// TwinCAT 3 PLC project Valve_AutoCalibration
// ProgramVersion: 3.1.4023.0
// libraries:
//   Tc2_Standard, * (Beckhoff Automation GmbH)
//   Tc2_System, * (Beckhoff Automation GmbH)
//   Tc3_Module, * (Beckhoff Automation GmbH)
// project tree:
//   / PlcTask.TcTTO
//   POUs/AutoCalibrate/ FB_AutoCalibration.TcPOU, FB_OnSetpointCheck.TcPOU, FB_PulseGen.TcPOU
//   POUs/ MAIN.TcPOU
// real-time tasks:
//   TASK PlcTask: cycle T#10ms, priority 20, ADS port 350

CONFIGURATION Valve_AutoCalibration
    RESOURCE PLC ON TwinCAT3
        TASK PlcTask(INTERVAL := T#10ms, PRIORITY := 20);
        PROGRAM MAIN WITH PlcTask : MAIN;
    END_RESOURCE
END_CONFIGURATION

// ---- POUs/MAIN.TcPOU
PROGRAM MAIN
VAR
bCalibrate:	BOOL;
fFB: REAL;
fStepValue: REAL :=0.5;
fDev: REAL := 0.1;	
fCmd: REAL;
fCommandZeroError:	REAL;
fCommandSpanError:	REAL;
fFeedbackZeroError:	REAL;
fFeedbackSpanError: REAL;  
bCalibrationFinished: BOOL;
bError : BOOL;
bBusy : BOOL;
bDoubleCheck : BOOL;
fbAutoCalibration : FB_AutoCalibration;
END_VAR

fbAutoCalibration(bCalibrate:=bCalibrate,
				fFB := fFB,
				fStepValue:=fStepValue,
				fDev:=fDev,
				fBand:=0.2);

fCmd:= fbAutoCalibration.fCmd;
				
fCommandZeroError:= fbAutoCalibration.fCmdZeroErr;

fCommandSpanError:= fbAutoCalibration.fCmdSpanErr;

fFeedbackZeroError:= fbAutoCalibration.fFBZeroErr;

fFeedbackSpanError:= fbAutoCalibration.fFBSpanErr;

bCalibrationFinished:=fbAutoCalibration.bCalibrationFinished;

bError := fbAutoCalibration.bError;

bBusy := fbAutoCalibration.bBusy;

bDoubleCheck := fbAutoCalibration.bDoubleCheck;

END_PROGRAM

// ---- POUs/AutoCalibrate/FB_AutoCalibration.TcPOU
FUNCTION_BLOCK FB_AutoCalibration
VAR_INPUT	
	bCalibrate:	BOOL; 	 //Calibration is ON
	fFB: REAL;			 //Valve feedback
	fStepValue: REAL;	 //Step value for the control valve
	fDev: REAL;			 //Deviation value to be catched in the feedback signal after the control valve stepped up
	fBand: REAL;		 //Acceptable deviation in the feedback for the double check
END_VAR
VAR_OUTPUT
	fCmd: REAL;					//Valve control signal
	fCmdZeroErr: REAL;			//Control singal zero error
	fCmdSpanErr: REAL;			//Control singal span error
	fFBZeroErr:	REAL;			//Feedback signal zero error
	fFBSpanErr: REAL;  			//Feedback span error	
	bCalibrationFinished: BOOL;	//Calibration completed
	bDoubleCheck: BOOL;			//True: Double check succesfful, FALSE: Double check failed 
	bBusy: BOOL;				//Calibration is working
	bError: BOOL;				//Error, if the valve does not open, close or exceeds the min/max values
END_VAR
VAR	
	bZeroErrCalibComplet: BOOL;
	bSpanErrCalibComplet: BOOL;
	fbPulseGenZeroErr : FB_PulseGen;
	fbPulseGenSpanErr : FB_PulseGen;
	fCmdPrevState : REAL;
	fFBPrevState : REAL;	
	RTrigCalibON : R_TRIG;	
	RTrigZero : R_TRIG;
	RTrigSpan : R_TRIG;
	bValveClosed : BOOL;
	bValveOpened : BOOL;
	bDoubleCheckFail  : BOOL;
	_fbTimerValveClosing: TON;
	_fbTimerValveOpening : TON;
	_bClosingTimer : BOOL;	
	_bOpeningTimer : BOOL;	
	_fbTimerDoubleCheck : TON;
	_bTimerDoubleCheck : BOOL;	
	_fbTimerOnMinFB	: TON;
	_fbTimerOnMaxFB	: TON;
	_bMinFBChecked : BOOL;
	_bMaxFBChecked : BOOL;
END_VAR
VAR CONSTANT
	fMinPos: REAL := 0.0;
	fMaxPos: REAL := 100.0;
	tPtON: TIME := T#0.01S;
	tPtOFF: TIME := T#5S;
	_tCloseValve: TIME := T#20S;		//20 seconds for closing the valve
	_tOpenValve: TIME := T#120S;		//120 seconds for opening the valve
	_fMinFB: REAL := 3.0;				//Min Input signal 4mA +- %2
	_fMaxFB: REAL := 96.04;				//Max Input signal 19.6mA +- %2
	_tDoubleCheck : TIME := T#150S;		//Max time for completing the double check (120s opening + 20s closing + 10s on FB check)	
	_tDelay : TIME := T#5S;				//Time for on setpoint check
END_VAR

//Initialization for the next calibration cycle
RTrigCalibON(CLK:= bCalibrate);
IF RTrigCalibON.Q AND NOT bBusy THEN		
	fFBPrevState := fFB;	
	fCmdZeroErr:= 0.0;
	fCmdSpanErr:= 0.0;
	fFBZeroErr:= 0.0;
	fFBSpanErr:= 0.0;
	bDoubleCheck:= FALSE;
	bDoubleCheckFail:= FALSE;
	bError := FALSE;	
	bBusy := TRUE;		
	bZeroErrCalibComplet := FALSE;
	bSpanErrCalibComplet := FALSE;
	bCalibrationFinished:= FALSE;	
	bValveClosed  := FALSE;
	bValveOpened  := FALSE;
	_bClosingTimer := TRUE;	
	_bOpeningTimer := FALSE;
	_bTimerDoubleCheck:= TRUE;	
	_bMinFBChecked := FALSE;
	_bMaxFBChecked := FALSE;
END_IF

//Zero error
CloseValve();
IF bValveClosed AND NOT bZeroErrCalibComplet THEN
	ZeroErrorCalibration();
END_IF

//Span error 	
OpenValve();
IF bValveOpened AND NOT bSpanErrCalibComplet THEN
	SpanErrorCalibration();
END_IF

//Double check	
IF bZeroErrCalibComplet AND bSpanErrCalibComplet THEN	
	DoubleCheck();			
END_IF

//Calibration completed
IF bDoubleCheck OR bDoubleCheckFail THEN
	bCalibrationFinished:= TRUE;	
	bBusy:= FALSE;	
ELSIF bError THEN	
	bCalibrationFinished:= FALSE;				
	bBusy:= FALSE;				
END_IF

METHOD CloseValve 
VAR_INPUT
END_VAR
_fbTimerValveClosing(IN:=_bClosingTimer,PT:=_tCloseValve);
IF NOT bValveClosed THEN
	fCmd:= fMinPos;
	IF _fbTimerValveClosing.Q AND (fFB < _fMinFB) THEN
		_bClosingTimer:=FALSE;
		bValveClosed := TRUE;		
	ELSIF _fbTimerValveClosing.Q AND NOT bValveClosed THEN		
		_bClosingTimer:=FALSE;	
		bError := TRUE;
	END_IF
END_IF
END_METHOD

METHOD DoubleCheck
VAR_INPUT
END_VAR
_fbTimerDoubleCheck(IN:=_bTimerDoubleCheck, PT:= _tDoubleCheck);
IF NOT _fbTimerDoubleCheck.Q THEN
	IF NOT _bMinFBChecked THEN
		fCmd:= fMinPos;
		IF fFB > (fFBZeroErr - fBand) AND fFB < (fFBZeroErr + fBand) THEN			
			_fbTimerOnMinFB(IN:=TRUE,PT:=_tDelay);				
		ELSE
			_fbTimerOnMinFB(IN:=FALSE);
		END_IF
		_bMinFBChecked:= _fbTimerOnMinFB.Q;
	ELSIF _bMinFBChecked AND NOT _bMaxFBChecked THEN
		fCmd:= fMaxPos;
		IF fFB > ((fMaxPos - fFBSpanErr) - fBand) AND fFB < ((fMaxPos - fFBSpanErr) + fBand) THEN			
			_fbTimerOnMaxFB(IN:=TRUE,PT:=_tDelay);	
		ELSE
			_fbTimerOnMaxFB(IN:=FALSE);
		END_IF
			_bMaxFBChecked:= _fbTimerOnMaxFB.Q;	
	ELSIF _bMinFBChecked AND _bMaxFBChecked THEN
			_bTimerDoubleCheck := FALSE;
			bDoubleCheck:= TRUE;
	END_IF	
ELSE
	_bTimerDoubleCheck := FALSE;	
	bDoubleCheckFail:= TRUE;
END_IF
END_METHOD

METHOD OpenValve 
VAR_INPUT
END_VAR
_fbTimerValveOpening(IN:=_bOpeningTimer,PT:=_tOpenValve);
IF NOT bValveOpened and bZeroErrCalibComplet THEN
	fCmd:= fMaxPos;
	IF _fbTimerValveOpening.Q AND (fFB >_fMaxFB) THEN		
		_bOpeningTimer:=FALSE;	
		bValveOpened:= TRUE;
	ELSIF _fbTimerValveOpening.Q AND NOT bValveOpened THEN
		_bOpeningTimer:=FALSE;	
		bError := TRUE;		
	END_IF	
END_IF
END_METHOD

METHOD SpanErrorCalibration
VAR_INPUT
END_VAR
fbPulseGenSpanErr(In:= NOT bSpanErrCalibComplet,Pt_ON:=tPtON, Pt_OFF:=tPtOFF);		
RTrigSpan(CLK:=fbPulseGenSpanErr.Q);
IF (fCmd <= fMinPos) THEN
	bError := TRUE;
ELSIF RTrigSpan.Q THEN
	fCmdPrevState:= fCmd;
	fFBPrevState:= fFB;
	fCmd := fCmd - fStepValue;
ELSIF (fFBPrevState - fFB >= fDev) THEN
	fCmdSpanErr:= fMaxPos - fCmdPrevState;
	fFBSpanErr:= fMaxPos - fFBPrevState;		
	bSpanErrCalibComplet:= TRUE;							
END_IF
END_METHOD

METHOD ZeroErrorCalibration
VAR_INPUT
END_VAR
fbPulseGenZeroErr(In:= NOT bZeroErrCalibComplet,Pt_ON:=tPtON, Pt_OFF:=tPtOFF);	  
RTrigZero(CLK:=fbPulseGenZeroErr.Q);
IF (fCmd >= fMaxPos) THEN
	bError := TRUE;
ELSIF RTrigZero.Q AND(fCmd <= fMaxPos) THEN
	fCmdPrevState := fCmd;
	fFBPrevState:= fFB;
	fCmd := fCmd + fStepValue;	
ELSIF(fFB - fFBPrevState >= fDev) THEN
	fCmdZeroErr:= fCmdPrevState;
	fFBZeroErr:= fFBPrevState;			
	bZeroErrCalibComplet:= TRUE;
	_bOpeningTimer := TRUE;			
END_IF
END_METHOD

END_FUNCTION_BLOCK

// ---- POUs/AutoCalibrate/FB_PulseGen.TcPOU
FUNCTION_BLOCK FB_PulseGen
    VAR_INPUT
        IN : BOOL;
        PT_ON : TIME;
        PT_OFF : TIME;
    END_VAR
    VAR_OUTPUT
		ET : TIME;
        Q : BOOL;        
    END_VAR
    VAR
        rtIN : R_TRIG;
        tonBlink : TON;
    END_VAR

rtIN(CLK := IN);
IF tonBlink.Q OR rtIN.Q THEN
    (*Toggle Output*)
    Q := NOT Q;    
    (*Timer Reset call, important to call timer twice in same cycle for correct Blink Time*)
    tonBlink(IN:= FALSE);    
    (*Set corresponding Time*)
    IF Q THEN
        tonBlink.PT := PT_ON;
    ELSE
        tonBlink.PT := PT_OFF;
    END_IF    
END_IF
(*Timer Run call*)
tonBlink(IN:= IN);

IF IN THEN
    ET := tonBlink.ET;
ELSE
    ET := T#0S;
    Q := FALSE;
END_IF

END_FUNCTION_BLOCK

// ---- POUs/AutoCalibrate/FB_OnSetpointCheck.TcPOU
FUNCTION_BLOCK FB_OnSetpointCheck
VAR_INPUT
	fSP			: REAL; 
	fFB			: REAL;	
	fBand		: REAL;	
	tDelay		: TIME;	
END_VAR
VAR_OUTPUT
	bOnSP	: BOOL := FALSE;
	fCmd	: REAL;	
END_VAR 
VAR
	fbTon	: TON;
END_VAR

fCmd := fSP;

IF fFB > (fSP - fBand) AND fFB < (fSP + fBand) THEN
	fbTon(IN := TRUE, PT := tDelay);
ELSE
	fbTon(IN := FALSE);
END_IF

bOnSP := fbTon.Q;

END_FUNCTION_BLOCK
